// TIA Portal V20 export
// export: Created 2025-12-01T14:57:23.5824636Z, ExportSetting None, DisplayName Totally Integrated Automation Portal, DisplayVersion V20 Update 3, DisplayName TIA Portal Openness, DisplayVersion V20 Update 3, DisplayName TIA Portal Version Control Interface, DisplayVersion V20 Update 3, DisplayName STEP 7 Professional, DisplayVersion V20 Update 3, DisplayName STEP 7 Safety, DisplayVersion V20 Update 2, DisplayName WinCC Basic/Comfort/Advanced, DisplayVersion V20 Update 3, DisplayName WinCC Professional, DisplayVersion V20 Update 3, DisplayName WinCC Unified, DisplayVersion V20 Update 3
DATA_BLOCK "DB1904_Datos_Config_Gateways"   // DB1904
{ S7_Optimized_Access := 'TRUE' }
// stored: AutoNumber false, MemoryReserve 100
   VAR RETAIN
      Gateway { ExternalAccessible := 'False'; ExternalVisible := 'False'; ExternalWritable := 'False'} : Array[1..16] of Struct
         Diagnosticar { S7_SetPoint := 'True'} : Bool;   // activar el diagnosticar solo si existe
         Dos_lineas { S7_SetPoint := 'True'} : Bool;
         hwld { S7_SetPoint := 'True'} : HW_INTERFACE;
         Dir_ini_diag { S7_SetPoint := 'True'} : Int;
         Dir_ini_Asi5_L1 { S7_SetPoint := 'True'} : Int;
         Dir_ini_ASi5_L2 { S7_SetPoint := 'True'} : Int;
      END_STRUCT;
   END_VAR
BEGIN
   Gateway[1].Diagnosticar := true;
   Gateway[1].Dos_lineas := true;
   Gateway[1].hwld := 276;
   Gateway[1].Dir_ini_diag := 6000;
   Gateway[1].Dir_ini_Asi5_L1 := 600;
   Gateway[1].Dir_ini_ASi5_L2 := 900;
END_DATA_BLOCK
